Staubli VAL3: Control_BatSpd.pgx

public program Control_BatSpd(num& x_nFrom, num& x_nTo, num& x_nSpeed, num& x_nAcc)
  local string l_sItem[4]
  local num l_nNum
  local num l_nKey
  local num l_nData[6]
  local num l_nSelectIndex
begin

  //为lasman3.0进行配置
  //批处理速度


  l_nData[0]=x_nFrom
  l_nData[1]=x_nTo
  l_nData[2]=100
  l_nData[3]=15
  l_sItem[0]="开始序号:"+toString("",l_nData[0])
  l_sItem[1]="结束序号:"+toString("",l_nData[1])
  l_sItem[2]="速度    :"+toString("",l_nData[2])
  l_sItem[3]="加速度  :"+toString("",l_nData[3])



  call Control_BottomS(",,,,,,取消,确定")
  call Control_PanelXY(8,0,15,4)
  call Control_Panel("批处理速度")
  call Control_List(l_sItem,l_nSelectIndex)
  while true
    l_nKey=getKey()

    switch l_nKey
      case 261
        l_nSelectIndex=max(0,l_nSelectIndex-1)
      break

      case 266
        l_nSelectIndex=min(l_nSelectIndex+1,3)
      break

      case 278
        x_nFrom=l_nData[0]
        x_nTo=l_nData[1]
        x_nSpeed=l_nData[2]
        x_nAcc=l_nData[3]
        cls()
        return
      break


      case 277,255

        cls()
        return
      break

      case 270

        call Float_Edit(l_nData[l_nSelectIndex],nPanelLTopX+7,l_nSelectIndex+nPanelLTopY+1)
      break

    endSwitch

    if l_nKey!=-1
  l_sItem[0]="开始序号:"+toString("",l_nData[0])
  l_sItem[1]="结束序号:"+toString("",l_nData[1])
  l_sItem[2]="速度    :"+toString("",l_nData[2])
  l_sItem[3]="加速度  :"+toString("",l_nData[3])
      call Control_List(l_sItem,l_nSelectIndex)

    endIf






  endWhile





end
